// TimeZone
fbSpecificLocalTime(in := Tc2_Utilities.FILETIME64_TO_SYSTEMTIME(fbEvent.nTimestamp), tzInfo := fbTimeZone.tzInfo, out => _TempTimestruct);

// Timestamp	
THIS^.stEventInfo.TimeRaised[0] := TO_DINT(_TempTimestruct.wYear);
THIS^.stEventInfo.TimeRaised[1] := TO_DINT(_TempTimestruct.wMonth);
THIS^.stEventInfo.TimeRaised[2] := TO_DINT(_TempTimestruct.wDay);
THIS^.stEventInfo.TimeRaised[3] := TO_DINT(_TempTimestruct.wHour);
THIS^.stEventInfo.TimeRaised[4] := TO_DINT(_TempTimestruct.wMinute);
THIS^.stEventInfo.TimeRaised[5] := TO_DINT(_TempTimestruct.wSecond);
THIS^.stEventInfo.TimeRaised[6] := TO_DINT(_TempTimestruct.wMilliseconds);
Tc2_System.MEMSET(destAddr := ADR(stEventInfo.TimeCleared), fillByte := 0, n := SIZEOF(stEventInfo.TimeCleared));
Tc2_System.MEMSET(destAddr := ADR(stEventInfo.TimeConfirmed), fillByte := 0, n := SIZEOF(stEventInfo.TimeConfirmed));

//store event info globally
aEventInfoBuffer[CntAlarmsRaised] := stEventInfo;

// activate requests in event triggered method 'OnMessageSent' to get related request info
aEventInfoBuffer[CntAlarmsRaised].fbRequestEventText.Request(eventClass := aEventInfoBuffer[CntAlarmsRaised].EventClass,
															 nEventId	:= aEventInfoBuffer[CntAlarmsRaised].EventId,
															 nLangId	:= 1033,
															 ipArgs		:= aEventInfoBuffer[CntAlarmsRaised].ipArguments);

OnAlarmRaised := S_OK; // in order to receive more callbacks (Set <> S_OK in order to cancel the callbacks for this program cycle.)
END_METHOD

PROPERTY ParentResponseDefinitions : ARRAY[0..4] OF SPT_BaseTypes.E_AlarmResponse
GET
ParentResponseDefinitions := _ParentResponseDefinitions;
END_GET
SET
_ParentResponseDefinitions := ParentResponseDefinitions;
END_SET
END_PROPERTY

METHOD Reset : BOOL
//This may or may not be called depending on the component type 

//which derives FB_ComponentBase
F_ClearAllEventsInClass(PackMLEventHandlerAlarms);
Reset := TRUE;
END_METHOD

METHOD PUBLIC TimeZone : BOOL
VAR_INST
	_Step : USINT; // Step Variable
END_VAR
CASE _Step OF
	0: // Start to get local Timezone 
		fbTimeZone.bExecute := TRUE;
		IF fbTimeZone.bBusy THEN
			_Step := _Step + 1;
		END_IF

	1: // set 
		fbTimeZone.bExecute := FALSE;
		_Step				:= 0;
		TimeZone			:= TRUE;

ELSE
	Tc2_System.ADSLOGSTR(msgCtrlMask := cMsgCtrlMask, msgFmtStr := Tc2_Standard.CONCAT(cBaseMsg, 'TimeZone: %s'), strArg := 'Case Idx error');
	_InternalError := TRUE;
END_CASE

fbTimeZone(sNetID := '');
IF fbTimeZone.bError THEN
	Tc2_System.ADSLOGSTR(msgCtrlMask := cMsgCtrlMask, msgFmtStr := Tc2_Standard.CONCAT(cBaseMsg, 'fbTimeZone ErrID: %s'), strArg := TO_STRING(fbTimeZone.nErrID));
	_InternalError := TRUE;
END_IF
END_METHOD

PROPERTY WarningToStopReason : BOOL
SET
_WarningToStopReason := WarningToStopReason;
END_SET
END_PROPERTY

METHOD PRIVATE WriteAlarmTags : HRESULT;
VAR_INPUT
	Alarm_Ref	  : REFERENCE TO Tc3_PackML_V2.ST_Alarm; // Reference to ST_Alarm of an new Alarm / Warning / Stop reason
	EventInfo_Ref : REFERENCE TO ST_EventInfo;			 // Reference to ST_EventInfo
	Trigger		  : BOOL;								 // Set / Reset Trigger in PML Structure
	AlarmIndex	  : DINT;								 // Alarm index
END_VAR
IF __ISVALIDREF(Alarm_Ref) AND __ISVALIDREF(EventInfo_Ref) THEN
	Alarm_Ref.ID	   := TO_DINT(EventInfo_Ref.EventId);
	Alarm_Ref.Value	   := AlarmIndex;
	Alarm_Ref.Message  := EventInfo_Ref.EventText;
	Alarm_Ref.Category := TO_DINT(EventInfo_Ref.eSeverity); // Verbose:=0, Info:=1, Warning:=2, Error:=3, Critical:=4
	Alarm_Ref.Trigger  := Trigger;
	Alarm_Ref.DateTime := EventInfo_Ref.TimeRaised;
	WriteAlarmTags	   := S_OK;
ELSE
	// Set internal Error
	Tc2_System.ADSLOGSTR(msgCtrlMask := cMsgCtrlMask, msgFmtStr := Tc2_Standard.CONCAT(cBaseMsg, 'WriteAlarmTags: %s'), strArg := 'Input-reference error');
	WriteAlarmTags := E_FAIL;
	_InternalError := TRUE;
END_IF
END_METHOD

END_FUNCTION_BLOCK

// Project Information/F_GetCompany
// This function has been automatically generated from the project information.
{attribute 'signature_flag' := '1073741824'}
{attribute 'TcGenerated'}
{attribute 'no-analysis'}
FUNCTION F_GetCompany : WSTRING
VAR_INPUT
	
END_VAR

F_GetCompany := "Beckhoff Automation LLC";

END_FUNCTION

// Project Information/F_GetTitle
// This function has been automatically generated from the project information.
{attribute 'signature_flag' := '1073741824'}
{attribute 'TcGenerated'}
{attribute 'no-analysis'}
FUNCTION F_GetTitle : WSTRING
VAR_INPUT
	
END_VAR

F_GetTitle := "SPT Components";

END_FUNCTION

// Project Information/F_GetVersion
// This function has been automatically generated from the project information.
{attribute 'signature_flag' := '1073741824'}
{attribute 'TcGenerated'}
{attribute 'no-analysis'}
FUNCTION F_GetVersion : ST_LibVersion
VAR_INPUT
	
END_VAR

F_GetVersion.iMajor := 3;
F_GetVersion.iMinor := 2;
F_GetVersion.iBuild := 3;
F_GetVersion.iRevision := 0;
F_GetVersion.sVersion := '3.2.3';
F_GetVersion.nFlags := 1;

END_FUNCTION

// Sensors/FB_DigitalSensor
FUNCTION_BLOCK FB_DigitalSensor EXTENDS FB_ComponentBase IMPLEMENTS I_DigitalSensorBase
VAR
	HardwareInput AT %I*		: BOOL;			  //Hardware input bit from the hysical sensor
	_DebounceMode				: E_DebounceMode; //Defines the debounce model that will filter the sensor's output to the program
	_DebounceTime				: TIME;			  //Time input parameter for use in Debounce functionality
	_Inverted					: BOOL;			  //Defines the output polarity of the sensor - a "TRUE" value will result in the signal of the sensor being inverted
	_SimulationInput			: BOOL;			  //Provides configuration input to the simulation functionality
	_SimulationTimebase			: UDINT;
	_SimulationMode				: E_SensorSimulationMode; //Defines the mode of operation for the simulation functionality of this component
	_TimeActive					: TIME;					  //Tracks the amount of time that the sensor has been in an active state
	_TimeInactive				: TIME;					  //Tracks the amount of time that the sensor has been in an inactive state
	_Active						: BOOL;
	TON_ActiveTimer				: Tc2_Standard.TON; //Tracks the amount of time that the sensor has been in an active state
	TON_InactiveTimer			: Tc2_Standard.TON; //Tracks the amount of time that the sensor has been in an inactive state
	TON_DebounceTimer			: Tc2_Standard.TON; //Utilized in the debounce implementation
	TP_DebounceTimer			: Tc2_Standard.TP;	//Utilized in the debounce implementation
	DigitalSensor_HMI			: ST_DigitalSensor_HMI;
	SimulationPulse1_TP			: Tc2_Standard.TP; //Pulse Timer for simulated sensor pulse generation
	SimulationPulse2_TP			: Tc2_Standard.TP; //Pulse Timer for simulated sensor pulse generation
	HMICommand_DigitalSensor_RT : R_TRIG;
END_VAR

METHOD PUBLIC CyclicLogic
VAR_INPUT
END_VAR
SUPER^.CyclicLogic();
IF _Simulate THEN
	CASE _SimulationMode OF
		E_SensorSimulationMode.InputDriven:
			_Active := _SimulationInput;

		E_SensorSimulationMode.Periodic:
			SimulationPulse1_TP(IN := NOT SimulationPulse2_TP.Q, PT := UDINT_TO_TIME(_SimulationTimebase));
			SimulationPulse2_TP(IN := NOT SimulationPulse1_TP.Q, PT := UDINT_TO_TIME(_SimulationTimebase));
			_Active := SimulationPulse2_TP.Q;
	END_CASE
ELSE
	_Active := ProcessInput(Input := HardwareInput);
END_IF
END_METHOD

PROPERTY Active : BOOL
GET
Active := _Active;
END_GET
END_PROPERTY

PROPERTY DebounceMode : E_DebounceMode
GET
DebounceMode := _DebounceMode;
END_GET
SET
_DebounceMode := DebounceMode;
END_SET
END_PROPERTY

PROPERTY DebounceTime : TIME
GET
DebounceTime := _DebounceTime;
END_GET
SET
_DebounceTime := DebounceTime;
END_SET
END_PROPERTY

PROPERTY Inverted : BOOL
GET
Inverted := _Inverted;
END_GET
SET
_Inverted := Inverted;
END_SET
END_PROPERTY

PROPERTY SimulationInput : BOOL
GET
SimulationInput := _SimulationInput;
END_GET
SET
_SimulationInput := SimulationInput;
END_SET
END_PROPERTY

PROPERTY SimulationMode : E_SensorSimulationMode
GET
SimulationMode := _SimulationMode;
END_GET
SET
_SimulationMode := SimulationMode;
END_SET
END_PROPERTY

PROPERTY SimulationTimeBase : UDINT
GET
SimulationTimeBase := _SimulationTimebase;
END_GET
SET
_SimulationTimeBase := SimulationTimebase;
END_SET
END_PROPERTY

PROPERTY TimeActive : TIME
GET
TimeActive := _TimeActive;
END_GET
END_PROPERTY

PROPERTY TimeInactive : TIME
GET
TimeInactive := _TimeInactive;
END_GET
END_PROPERTY

METHOD PROTECTED HMICommunication
//Extend this method in extended FBs to communicate specific implementation data
SUPER^.HMICommunication();

//Process HMI requests

//Replace 'FALSE' below with further momentary commands (myCommand XOR myOtherCommand XOR...)
HMICommand_DigitalSensor_RT(CLK := (ComponentBase_HMI.Status.HMIControlAvailable AND NOT HMICommandActive_Base) AND (FALSE));

//Signal to FB_ComponentBase that a command is active
HMICommandActive_Descendant := ComponentBase_HMI.Status.HMIControlAvailable AND (DigitalSensor_HMI.Config.DebounceMode <> _DebounceMode OR DigitalSensor_HMI.Config.DebounceTime <> _DebounceTime OR DigitalSensor_HMI.Config.Inverted <> _Inverted OR DigitalSensor_HMI.Config.SimulationMode <> _SimulationMode OR DigitalSensor_HMI.Config.SimulationTimebase <> _SimulationTimebase);

//Process HMI requests
IF HMICommand_DigitalSensor_RT.Q THEN //If a request has been issued by the HMI, and a previous request has not just finished being processed

	//	IF AxisBaseHMI.Command.xxx THEN

	//		Enabled := TRUE;

	//	END_IF
END_IF

IF ComponentBase_HMI.Status.HMIControlAvailable AND NOT HMICommand_DigitalSensor_RT.Q THEN
	IF DigitalSensor_HMI.Config.DebounceMode <> _DebounceMode THEN
		DebounceMode := DigitalSensor_HMI.Config.DebounceMode;
	END_IF

	IF DigitalSensor_HMI.Config.DebounceTime <> _DebounceTime THEN
		DebounceTime := DigitalSensor_HMI.Config.DebounceTime;
	END_IF

	IF DigitalSensor_HMI.Config.Inverted <> _Inverted THEN
		Inverted := DigitalSensor_HMI.Config.Inverted;
	END_IF

	IF DigitalSensor_HMI.Config.SimulationMode <> _SimulationMode THEN
		SimulationMode := DigitalSensor_HMI.Config.SimulationMode;
	END_IF

	IF DigitalSensor_HMI.Config.SimulationTimebase <> _SimulationTimebase THEN
		SimulationTimeBase := DigitalSensor_HMI.Config.SimulationTimebase;
	END_IF
END_IF

//Update HMI status info
DigitalSensor_HMI.Status.Active				:= _Active;
DigitalSensor_HMI.Status.TimeActive			:= TIME_TO_LREAL(_TimeActive) / 1000.0;
DigitalSensor_HMI.Status.TimeInactive		:= TIME_TO_LREAL(_TimeInactive) / 1000.0;
DigitalSensor_HMI.Config.DebounceMode		:= DebounceMode;
DigitalSensor_HMI.Config.DebounceTime		:= DebounceTime;
DigitalSensor_HMI.Config.Inverted			:= Inverted;
DigitalSensor_HMI.Config.SimulationMode		:= SimulationMode;
DigitalSensor_HMI.Config.SimulationTimebase := SimulationTimeBase;
END_METHOD

METHOD PROTECTED Monitoring
SUPER^.Monitoring();

//If flicker counters or other diagnostic systems are desired, their implementation could be here

//Any warnings, errors, or other desired messages would also be generated here

//T#71582M47S295MS is the upper bound of the TIME type, meaning these timers will continue to increase ET for as long as possible
TON_ActiveTimer(IN := _Active, PT := T#71582M47S295MS, ET => _TimeActive);
TON_InactiveTimer(IN := NOT _Active, PT := T#71582M47S295MS, ET => _TimeInactive);
_Busy  := FALSE;
_Error := FALSE;
END_METHOD

METHOD PRIVATE ProcessInput : BOOL
VAR_INPUT
	Input : BOOL;
END_VAR

VAR
	DebouncedInput : BOOL;
END_VAR

VAR_INST
	LastDebouncedInput : BOOL;
	MovingAverage	   : DINT;
END_VAR
CASE DebounceMode OF
	E_DebounceMode.RawInput: //Passes raw input through
		DebouncedInput := Input;

	E_DebounceMode.SimpleFlickerFilter:											 //Requires the raw input to be a consistent value for a set time period before output changes
		TON_DebounceTimer(IN := (Input <> DebouncedInput), PT := _DebounceTime); //runs the timer whenever a differing input is detected
		IF TON_DebounceTimer.Q THEN
			DebouncedInput := Input; //once the raw input has been different for the specified debounce time, the processed input is updated
		END_IF

	E_DebounceMode.EdgeDetectFilter:								   //Updates the processed value immediately on a change from steady state, but mutes any sensor flickers for the specified time immediately following the change
		IF (Input <> DebouncedInput) AND (NOT TP_DebounceTimer.Q) THEN //A differing raw input must be detected outside of the mute window created by the pulse timer
			DebouncedInput := Input;
		END_IF

		TP_DebounceTimer(IN := (DebouncedInput <> LastDebouncedInput), PT := _DebounceTime); //"Q" will be TRUE for tDebounce time after the bProcessedSensorInput value is changed
	E_DebounceMode.MovingAverage:															 //Uses a "moving average"-like calculation to compensate for extremely inconsistent signals - prevents poorly timed flickers from causing disproportionate results
		TON_DebounceTimer(IN := NOT TON_DebounceTimer.Q, PT := T#5MS);						 //Provides a 1ms "polling" trigger
		IF TON_DebounceTimer.Q THEN															 //TRUE once every millisecond
			IF Input THEN																	 //If raw input is currently active at the time of polling
				IF MovingAverage < TIME_TO_DINT(_DebounceTime) THEN							 //If the moving average has not reached its "weight limit" as set by debounce time
					MovingAverage := MovingAverage + 5;										 //Add 1 to the average
				END_IF
			ELSE													 //If raw input is currently inactive at the time of polling
				IF MovingAverage > -TIME_TO_DINT(_DebounceTime) THEN //If the moving average has not reached its "weight limit" as set by debounce time
					MovingAverage := MovingAverage - 5;				 //Subtract 1 from the average
				END_IF
			END_IF
		END_IF

		IF MovingAverage >= 0 THEN
			DebouncedInput := TRUE;
		ELSE
			DebouncedInput := FALSE;
		END_IF
END_CASE

LastDebouncedInput := DebouncedInput; //Update "Last value"
IF _Inverted THEN					  //If signal inversion is requested, invert the signal
	DebouncedInput := NOT DebouncedInput;
END_IF

ProcessInput := DebouncedInput;
END_METHOD

END_FUNCTION_BLOCK

// Sensors/I_DigitalSensorBase
INTERFACE I_DigitalSensorBase

PROPERTY DebounceMode : E_DebounceMode
GET
END_GET
SET
END_SET
END_PROPERTY

PROPERTY DebounceTime : TIME
GET
END_GET
SET
END_SET
END_PROPERTY

PROPERTY Inverted : BOOL //"High" signal from the sensor will be interpreted as an "inactive" reading when this parameter is TRUE
GET
END_GET
SET
END_SET
END_PROPERTY

PROPERTY SimulationInput : BOOL
GET
END_GET
SET
END_SET
END_PROPERTY

PROPERTY SimulationMode : E_SensorSimulationMode
GET
END_GET
SET
END_SET
END_PROPERTY

PROPERTY TimeActive : TIME
GET
END_GET
END_PROPERTY

PROPERTY TimeInactive : TIME
GET
END_GET
END_PROPERTY

END_INTERFACE

// Solenoids/SolenoidBankBase/FB_SolenoidBankBase
FUNCTION_BLOCK ABSTRACT FB_SolenoidBankBase EXTENDS FB_ComponentBase
VAR
	// Configuration
	Configuration : ARRAY[1..Parameters_Cylinder.MAX_NUMBER_OF_SOLENOIDS] OF ST_SolenoidBankConfig;

	//Counted number of solenoids
	NumberOfSolenoids : UINT;

	//Alarms
	SolenoidBankAlarms : ARRAY[1..SolenoidBankBaseAlarmsCount] OF FB_TcAlarm;
END_VAR

VAR CONSTANT
	SolenoidBankBaseAlarmsCount : UINT := 2;
END_VAR

METHOD PUBLIC AddSolenoid : UINT
VAR_INPUT
	ipCylinder	 : I_Solenoid;
	Number		 : UINT; //This is the number in the IO tree.
	SolenoidType : E_SolenoidType;
END_VAR
IF CheckNumber(Number) AND ipCylinder <> 0 THEN
	NumberOfSolenoids									  := NumberOfSolenoids + 1;
	Configuration[NumberOfSolenoids].ipSolenoid			  := ipCylinder;
	Configuration[NumberOfSolenoids].SolenoidType		  := SolenoidType;
	Configuration[NumberOfSolenoids].SolenoidOutputNumber := Number;
END_IF
END_METHOD

METHOD PRIVATE CheckNumber : BOOL
VAR_INPUT
	Number : UINT;
END_VAR
CheckNumber := TRUE;
IF Number < 1 AND Number > Parameters_Cylinder.MAX_NUMBER_OF_SOLENOIDS THEN
	IF NOT SolenoidBankAlarms[E_CylinderBankAlarms.CylinderNumberOutOfRange].bRaised THEN
		SolenoidBankAlarms[E_CylinderBankAlarms.CylinderNumberOutOfRange].Raise(0);
	END_IF

	CheckNumber := FALSE;
END_IF
END_METHOD

//! @summary Initializes event function blocks using this components's name
{attribute 'call_after_online_change_slot' := '<slot>'}
METHOD PROTECTED CreateEvents

//! @description This method is called by <c>Initialize()</c> as required
SUPER^.CreateEvents();
F_CreateAllEventsInClass(Alarms		:= SolenoidBankAlarms,
						 ClassSize	:= SIZEOF(TC_EVENTS.CylinderBankAlarms),
						 pInitEvent := ADR(TC_EVENTS.CylinderBankAlarms.InitReferenceEvent),
						 Prefix		:= Name);
END_METHOD

//! @summary This method serves as the entry point for all underlying FB logic
METHOD PUBLIC CyclicLogic
//! @description This method should be called cyclically by descendant function blocks by invoking <c>SUPER^.CyclicLogic()</c>.  Alternatively, the contents of this method could be reimplemented entirely in which case a call to this method would not be necessary.
VAR
	x : UINT;
END_VAR
//Loop through all solenoids that are added.
FOR x := 1 TO NumberOfSolenoids DO
	MapIO(x);
END_FOR
END_METHOD

//! @summary Basic component initialization logic
METHOD PROTECTED Initialize : BOOL;
//! @description This method is called by <c>CyclicLogic()</c> as required
VAR
	x : UINT;
END_VAR
NumberOfSolenoids := 0;
Initialize		  := TRUE;
END_METHOD

METHOD ABSTRACT MapIO
VAR_INPUT
	x : UINT;
END_VAR
END_METHOD

//! Provides basic error detection and event handling for this component
METHOD PROTECTED Monitoring

(*! @descriptionThis method is called cyclically by <c>CyclicLogic()</c>*)
SUPER^.Monitoring();
_CurrentAlarmSeverity := F_GetMaxSeverityRaised(Alarms := SolenoidBankAlarms, CurrentSeverity := CurrentAlarmSeverity);
END_METHOD

//! @summary Clears error flags and error IDs for this component
METHOD PUBLIC Reset : BOOL
SUPER^.Reset();
IF SolenoidBankAlarms[E_CylinderBankAlarms.CylinderNumberOutOfRange].bRaised THEN
	SolenoidBankAlarms[E_CylinderBankAlarms.CylinderNumberOutOfRange].Clear(0, 0);
END_IF
END_METHOD

END_FUNCTION_BLOCK

// Solenoids/I_Solenoid
INTERFACE I_Solenoid

METHOD Extend
VAR_INPUT
END_VAR
END_METHOD

PROPERTY Extended : BOOL
GET
END_GET
END_PROPERTY

PROPERTY ExtendOutput : BOOL
GET
END_GET
END_PROPERTY

PROPERTY ExtendTime : LREAL
GET
END_GET
SET
END_SET
END_PROPERTY

METHOD Retract
VAR_INPUT
END_VAR
END_METHOD

PROPERTY Retracted : BOOL
GET
END_GET
END_PROPERTY

PROPERTY RetractOutput : BOOL
GET
END_GET
END_PROPERTY

PROPERTY RetractTime : LREAL
GET
END_GET
SET
END_SET
END_PROPERTY

END_INTERFACE

// Solenoids/FB_DoubleSolenoid
FUNCTION_BLOCK FB_DoubleSolenoid EXTENDS FB_SingleSolenoid
VAR
	_RetractOutput AT %Q* : BOOL;
END_VAR

METHOD PROTECTED HardwareInit
//Update the status based on the IO 
IF _ExtendOutput AND NOT _RetractOutput THEN
	_Extended  := TRUE;
	_Retracted := FALSE;
ELSIF NOT _ExtendOutput AND _RetractOutput THEN
	_Extended  := FALSE;
	_Retracted := TRUE;
ELSE // By Default, set RetractOuptupt if neither is set or if both are set.
	_ExtendOutput  := FALSE;
	_RetractOutput := TRUE;
	_Extended	   := FALSE;
	_Retracted	   := TRUE;
END_IF
END_METHOD

METHOD PROTECTED HardwareUpdate
//One shot the requests
Extend_RTRIG(CLK := _ExtendRequest);
Retract_RTRIG(CLK := _RetractRequest);

//Handle Extend
IF Extend_RTRIG.Q THEN
	_ExtendOutput	:= TRUE;
	_RetractOutput	:= FALSE;
	_Extending		:= TRUE;
	_Retracting		:= FALSE;
	_Retracted		:= FALSE;
	_RetractRequest := FALSE;
END_IF

//Handle Retract
IF Retract_RTRIG.Q THEN
	_ExtendOutput  := FALSE;
	_RetractOutput := TRUE;
	_Extending	   := FALSE;
	_Retracting	   := TRUE;
	_Extended	   := FALSE;
	_ExtendRequest := FALSE;
END_IF

//Always Simulate Feedback here with no feedback inputs
Feedback();
END_METHOD

PROPERTY RetractOutput : BOOL
GET
RetractOutput := _RetractOutput;
END_GET
END_PROPERTY

END_FUNCTION_BLOCK

// Solenoids/FB_SingleSolenoid
(*	This FB is used for a single output solenoid 
	It uses the times to say when Extended/Retracted  	
	It starts assuming retracted and the output off.
*)
FUNCTION_BLOCK FB_SingleSolenoid EXTENDS FB_ComponentBase IMPLEMENTS I_Solenoid
VAR
	//Output
	_ExtendOutput AT %Q* : BOOL;

	// Internal variables
	_ExtendRequest	: BOOL;
	_RetractRequest : BOOL;
	_Extended		: BOOL;
	_Retracted		: BOOL;
	_Extending		: BOOL;
	_Retracting		: BOOL;
	_ExtendTime		: LREAL := 1000; // Default time 1s
	_RetractTime	: LREAL := 1000; // Default time 1s

	// Timer for Extend/Retract
	Extend_TON	  : TON;
	Retract_TON	  : TON;
	Extend_RTRIG  : R_TRIG;
	Retract_RTRIG : R_TRIG;

	//HMI 
	SolenoidHMI : ST_Cylinder_HMI;

	//Alarms
	SolenoidAlarms : ARRAY[1..SolenoidAlarmsCount] OF FB_TcAlarm;
END_VAR

VAR CONSTANT
	SolenoidAlarmsCount : UINT := 4;
END_VAR

METHOD PROTECTED CreateEvents
VAR_INPUT
END_VAR
SUPER^.CreateEvents();
F_CreateAllEventsInClass(Alarms		:= SolenoidAlarms,
						 ClassSize	:= SIZEOF(TC_EVENTS.CylinderAlarms),
						 pInitEvent := ADR(TC_EVENTS.CylinderAlarms.InitReferenceEvent),
						 Prefix		:= Name);
END_METHOD

METHOD PROTECTED HMICommunication
VAR_INPUT
END_VAR
SUPER^.HMICommunication();

//Handle the requests to extend and retract
IF ComponentBase_HMI.Status.HMIControlAvailable THEN
	IF SolenoidHMI.Command.Extend THEN
		Extend();
	ELSIF SolenoidHMI.Command.Retract THEN
		Retract();
	END_IF

	IF NOT F_CompareLREAL(SolenoidHMI.Command.ExtendTime, _ExtendTime, 0.01) THEN
		_ExtendTime := SolenoidHMI.Command.ExtendTime;
	END_IF

	IF NOT F_CompareLREAL(SolenoidHMI.Command.RetractTime, _RetractTime, 0.01) THEN
		_RetractTime := SolenoidHMI.Command.RetractTime;
	END_IF
END_IF

//Update HMI status info
SolenoidHMI.Status.Extended	   := _Extended;
SolenoidHMI.Status.Extending   := _Extending;
SolenoidHMI.Status.Retracted   := _Retracted;
SolenoidHMI.Status.Retracting  := _Retracting;
SolenoidHMI.Config.ExtendTime  := _ExtendTime;
SolenoidHMI.Config.RetractTime := _RetractTime;
END_METHOD

METHOD PROTECTED Monitoring
VAR_INPUT
END_VAR
SUPER^.Monitoring();

//Update output bits
_Busy				  := _Extending OR _Retracting;
_CurrentAlarmSeverity := F_GetMaxSeverityRaised(Alarms := SolenoidAlarms, CurrentSeverity := CurrentAlarmSeverity);
_Error				  := _CurrentAlarmSeverity >= TcEventSeverity.Error;
END_METHOD

METHOD CyclicLogic
VAR
	myErrorID : UDINT;
END_VAR
HardwareUpdate();
SUPER^.CyclicLogic();

//New code
myErrorID := THIS^.ErrorID;
END_METHOD

METHOD Extend
_ExtendRequest	:= TRUE;
_RetractRequest := FALSE;
END_METHOD

PROPERTY Extended : BOOL
GET
Extended := _Extended;
END_GET
END_PROPERTY

PROPERTY ExtendOutput : BOOL
GET
ExtendOutput := _ExtendOutput;
END_GET
END_PROPERTY

PROPERTY ExtendTime : LREAL
GET
ExtendTime := _ExtendTime;
END_GET
SET
_ExtendTime					   := ExtendTime;
SolenoidHMI.Command.ExtendTime := ExtendTime;
END_SET
END_PROPERTY

METHOD Retract
_ExtendRequest	:= FALSE;
_RetractRequest := TRUE;
END_METHOD

PROPERTY Retracted : BOOL
GET
Retracted := _Retracted;
END_GET
END_PROPERTY

PROPERTY RetractOutput : BOOL
GET
RetractOutput := FALSE;
END_GET
END_PROPERTY

PROPERTY RetractTime : LREAL
GET
RetractTime := _RetractTime;
END_GET
SET
_RetractTime					:= RetractTime;
SolenoidHMI.Command.RetractTime := RetractTime;
END_SET
END_PROPERTY

METHOD PROTECTED Feedback
VAR_INPUT
END_VAR
//Handle the time to Extend/Retract
Extend_TON(IN := _Extending, PT := LREAL_TO_TIME(_ExtendTime));
Retract_TON(IN := _Retracting, PT := LREAL_TO_TIME(_RetractTime));
IF Extend_TON.Q THEN
	_Extended  := TRUE;
	_Extending := FALSE;
END_IF

IF Retract_TON.Q THEN
	_Retracted	:= TRUE;
	_Retracting := FALSE;
END_IF
END_METHOD

METHOD PROTECTED HardwareInit
IF _ExtendOutput THEN
	_Extended  := TRUE;
	_Retracted := FALSE;
ELSE
	_Extended  := FALSE;
	_Retracted := TRUE;
END_IF
END_METHOD

METHOD PROTECTED HardwareUpdate
VAR_INPUT
END_VAR
//One shot the requests
Extend_RTRIG(CLK := _ExtendRequest);
Retract_RTRIG(CLK := _RetractRequest);

//Handle Extend
IF Extend_RTRIG.Q THEN
	_ExtendOutput	:= TRUE;
	_Extending		:= TRUE;
	_Retracting		:= FALSE;
	_Retracted		:= FALSE;
	_RetractRequest := FALSE;
END_IF

//Handle Retract
IF Retract_RTRIG.Q THEN
	_ExtendOutput  := FALSE;
	_Extending	   := FALSE;
	_Retracting	   := TRUE;
	_Extended	   := FALSE;
	_ExtendRequest := FALSE;
END_IF

//Call the feedback 
Feedback();
END_METHOD

//! @summary Basic component initialization logic
METHOD PROTECTED Initialize : BOOL;

//! @description This method is called by <c>CyclicLogic()</c> as required
//Set the cylinder to retracted
_Extending		:= FALSE;
_ExtendRequest	:= FALSE;
_Retracting		:= FALSE;
_RetractRequest := FALSE;

//Set the HMI time to the currnt time.
SolenoidHMI.Command.ExtendTime	:= _ExtendTime;
SolenoidHMI.Command.RetractTime := _RetractTime;

//Call base class Initialize
Initialize := SUPER^.Initialize();

// Call the HardwareInit
HardwareInit();
END_METHOD

//! @summary Clears error flags and error IDs for this component
METHOD PUBLIC Reset : BOOL
Reset := FALSE;
F_ClearAllEventsInClass(Alarms := SolenoidAlarms);
END_METHOD

END_FUNCTION_BLOCK

// Solenoids/FB_DoubleSolenoidFeedback
FUNCTION_BLOCK FB_DoubleSolenoidFeedback EXTENDS FB_DoubleSolenoid
VAR
	ExtendedSensor	AT %I* : BOOL;
	RetractedSensor AT %I* : BOOL;
END_VAR

PROPERTY ExtendedInput : BOOL
SET
ExtendedSensor := ExtendedInput;
END_SET
END_PROPERTY

METHOD PROTECTED Feedback
IF NOT _Simulate THEN
	_Extended  := ExtendedSensor;
	_Retracted := RetractedSensor;
	Extend_TON(IN := _Extending, PT := LREAL_TO_TIME(_ExtendTime));
	Retract_TON(IN := _Retracting, PT := LREAL_TO_TIME(_RetractTime));
	IF Extend_TON.Q AND NOT ExtendedSensor THEN
		IF NOT SolenoidAlarms[E_CylinderAlarms.ExtendTimeout].bRaised THEN
			SolenoidAlarms[E_CylinderAlarms.ExtendTimeout].Raise(0);
			_ExtendRequest := FALSE;
			_Extending	   := FALSE;
		END_IF
	ELSIF _Extending AND ExtendedSensor THEN
		_Extended  := TRUE;
		_Extending := FALSE;
	END_IF

	IF Retract_TON.Q AND NOT RetractedSensor THEN
		IF NOT SolenoidAlarms[E_CylinderAlarms.RetractTimeout].bRaised THEN
			SolenoidAlarms[E_CylinderAlarms.RetractTimeout].Raise(0);
			_RetractRequest := FALSE;
			_Retracting		:= FALSE;
		END_IF
	ELSIF _Retracting AND RetractedSensor THEN
		_Retracted	:= TRUE;
		_Retracting := FALSE;
	END_IF
ELSE
	SUPER^.Feedback();
END_IF

//Monitor Inputs in case both on at the same time
IF ExtendedSensor AND RetractedSensor AND NOT SolenoidAlarms[E_CylinderAlarms.ExtendedAndRetracted].bRaised THEN
	SolenoidAlarms[E_CylinderAlarms.ExtendedAndRetracted].Raise(0);
ELSIF (ExtendedSensor XOR RetractedSensor) AND SolenoidAlarms[E_CylinderAlarms.ExtendedAndRetracted].bRaised THEN
	SolenoidAlarms[E_CylinderAlarms.ExtendedAndRetracted].Clear(0, 0);
END_IF
END_METHOD

METHOD PROTECTED HardwareInit
IF ExtendedSensor AND NOT RetractedSensor THEN
	_Extended  := TRUE;
	_Retracted := FALSE;
ELSIF NOT ExtendedSensor AND RetractedSensor THEN
	_Extended  := FALSE;
	_Retracted := TRUE;
ELSE // With Neither on, then this means that it is not either or maybe no air
	_Extended  := FALSE;
	_Retracted := FALSE;
END_IF
END_METHOD

PROPERTY RetractedInput : BOOL
SET
RetractedSensor := RetractedInput;
END_SET
END_PROPERTY

END_FUNCTION_BLOCK

// Solenoids/FB_SingleSolenoidFeedback
FUNCTION_BLOCK FB_SingleSolenoidFeedback EXTENDS FB_SingleSolenoid
VAR
	ExtendedSensor	AT %I* : BOOL;
	RetractedSensor AT %I* : BOOL;
END_VAR

PROPERTY ExtendedInput : BOOL
SET
ExtendedSensor := ExtendedInput;
END_SET
END_PROPERTY

METHOD PROTECTED Feedback
IF NOT _Simulate THEN
	_Extended  := ExtendedSensor;
	_Retracted := RetractedSensor;
	Extend_TON(IN := _Extending, PT := LREAL_TO_TIME(_ExtendTime));
	Retract_TON(IN := _Retracting, PT := LREAL_TO_TIME(_RetractTime));
	IF Extend_TON.Q AND NOT ExtendedSensor THEN
		IF NOT SolenoidAlarms[E_CylinderAlarms.ExtendTimeout].bRaised THEN
			SolenoidAlarms[E_CylinderAlarms.ExtendTimeout].Raise(0);
			_ExtendRequest := FALSE;
			_Extending	   := FALSE;
		END_IF
	ELSIF _Extending AND ExtendedSensor THEN
		_Extended  := TRUE;
		_Extending := FALSE;
	END_IF

	IF Retract_TON.Q AND NOT RetractedSensor THEN
		IF NOT SolenoidAlarms[E_CylinderAlarms.RetractTimeout].bRaised THEN
			SolenoidAlarms[E_CylinderAlarms.RetractTimeout].Raise(0);
			_RetractRequest := FALSE;
			_Retracting		:= FALSE;
		END_IF
	ELSIF _Retracting AND RetractedSensor THEN
		_Retracted	:= TRUE;
		_Retracting := FALSE;
	END_IF
ELSE
	SUPER^.Feedback(); //Call the feedback that usese timers for feedback
END_IF

//Monitor Inputs in case both on at the same time
IF ExtendedSensor AND RetractedSensor AND NOT SolenoidAlarms[E_CylinderAlarms.ExtendedAndRetracted].bRaised THEN
	SolenoidAlarms[E_CylinderAlarms.ExtendedAndRetracted].Raise(0);
ELSIF (ExtendedSensor XOR RetractedSensor) AND SolenoidAlarms[E_CylinderAlarms.ExtendedAndRetracted].bRaised THEN
	SolenoidAlarms[E_CylinderAlarms.ExtendedAndRetracted].Clear(0, 0);
END_IF
END_METHOD

METHOD PROTECTED HardwareInit
IF ExtendedSensor AND NOT RetractedSensor THEN
	_Extended  := TRUE;
	_Retracted := FALSE;
ELSIF NOT ExtendedSensor AND RetractedSensor THEN
	_Extended  := FALSE;
	_Retracted := TRUE;
ELSE // With Neither on, then this means that it is not either or maybe no air
	_Extended  := FALSE;
	_Retracted := FALSE;
END_IF
END_METHOD

PROPERTY RetractedInput : BOOL
SET
RetractedSensor := RetractedInput;
END_SET
END_PROPERTY

END_FUNCTION_BLOCK

// Testing/Axis/FB_ComponentBasicAxis_Test
FUNCTION_BLOCK FB_ComponentBasicAxis_Test EXTENDS TCUnit.FB_TestSuite
VAR
	TestFBInit					: FB_Component_BasicAxis;
	TestFBNameSetProperty		: FB_Component_BasicAxis;
	TestFBSimulationSetProperty : FB_Component_BasicAxis;
	TestFBSimulationSetHMI		: FB_Component_BasicAxis;
	TestFBSimulationCheckAlarm	: FB_Component_BasicAxis;
	TestFBBusy					: FB_Component_BasicAxis;
	TestFBAllowHMI				: FB_Component_BasicAxis;
	TestFBBlockHMI				: FB_Component_BasicAxis;

	//Axis integration test - this should be tested in the NCAxis library. (Enable, Disable, etc....)

	//Alarm Testing - 17 Alarms with FB_ComponentBasicAxis

	///TestFBAlarm1  FB_Component_BasicAxis; // InitReference (Not an actual alarm)
	TestFBAlarm2 : FB_Component_BasicAxis; // MC_Power
	TestFBAlarm3 : FB_Component_BasicAxis; // MC_Reset
	TestFBAlarm4 : FB_Component_BasicAxis; // MC_Halt

	///TestFBAlarm5 FB_Component_BasicAxis; // MC_Stop // Not Implemented
	TestFBAlarm6  : FB_Component_BasicAxis; // MC_Home
	TestFBAlarm7  : FB_Component_BasicAxis; // MC_Jog
	TestFBAlarm8  : FB_Component_BasicAxis; // MC_MoveAbsolute
	TestFBAlarm9  : FB_Component_BasicAxis; // MC_MoveRelative
	TestFBAlarm10 : FB_Component_BasicAxis; // MC_MoveVelocity
	TestFBAlarm11 : FB_Component_BasicAxis; // MC_MoveModulo
	TestFBAlarm12 : FB_Component_BasicAxis; // MC_ReadParameter
	TestFBAlarm13 : FB_Component_BasicAxis; // MC_WriteParameter
	TestFBAlarm14 : FB_Component_BasicAxis; // MC_WriteBOOLParameter
	TestFBAlarm15 : FB_Component_BasicAxis; // Command While Inhibited

	///TestFBAlarm16 FB_Component_BasicAxis; // Axis Error (Not Sure how to get Axis error with virtual axis)

	///TestFBAlarm17 FB_Component_BasicAxis; // Drive Error (Cannot Get Drive Error without drive)
END_VAR

Init();
NameSetProperty();
SimulationSetProperty();
SimulationSetHMI();
SimulationCheckAlarm();
Busy();
AllowHMI();
BlockHMI();

//Tests for Alarms
MCPowerAlarm();
MCResetAlarm();
MCHaltAlarm();
MCHomeAlarm();
MCJogAlarm();
MCMoveAbsoluteAlarm();
MCMoveRelativeAlarm();
MCMoveVelocity();
MCMoveModulo();
McReadAxisParametersAlarm();
McWriteAxisParameterAlarm();
McWriteAxisBoolParameterAlarm();
CommandInhibited();

METHOD AllowHMI
VAR_INST
	State		   : INT;
	ActualResult   : BOOL;
	ExpectedResult : BOOL := TRUE;
END_VAR
IF TEST_ORDERED('BasicAxisAllowHMI') THEN
	CASE State OF
		0:
			State := State + 10;

		10:
			IF TestFBAllowHMI.InitComplete AND NOT TestFBAllowHMI.Busy THEN
				TestFBAllowHMI.AllowHMIControl();
				State := State + 10;
			END_IF

		20:
			ActualResult := TestFBAllowHMI.ComponentBase_HMI.Status.HMIControlAvailable;
			AssertEquals_BOOL(Expected := ExpectedResult, Actual := ActualResult, Message := 'Function Block read allow HMI Control in HMI Tag not true');
			TEST_FINISHED();
			State := State + 10;
	END_CASE

	//Call to FB Cyclic Logic
	TestFBAllowHMI.CyclicLogic();
END_IF
END_METHOD

METHOD BlockHMI
VAR_INST
	State		   : INT;
	ActualResult   : BOOL;
	ExpectedResult : BOOL := FALSE;
END_VAR
IF TEST_ORDERED('BasicAxisBlockHMI') THEN
	CASE State OF
		0:
			State := State + 10;

		10:
			IF TestFBBlockHMI.InitComplete AND NOT TestFBBlockHMI.Busy THEN
				TestFBBlockHMI.AllowHMIControl();
				State := State + 10;
			END_IF

		20:
			IF TestFBBlockHMI.ComponentBase_HMI.Status.HMIControlAvailable THEN
				TestFBBlockHMI.BlockHMIControl();
				State := State + 10;
			END_IF

		30:
			ActualResult := TestFBBlockHMI.ComponentBase_HMI.Status.HMIControlAvailable;
			AssertEquals_BOOL(Expected := ExpectedResult, Actual := ActualResult, Message := 'Function Block read Block HMI Control in HMI Tag not false');
			TEST_FINISHED();
			State := State + 10;
	END_CASE

	//Call to FB Cyclic Logic
	TestFBBlockHMI.CyclicLogic();
END_IF
END_METHOD

METHOD Busy
VAR_INST
	State		   : INT;
	ActualResult   : BOOL;
	ExpectedResult : BOOL := TRUE;
	Timeout		   : TON;
END_VAR
IF TEST_ORDERED('BasicAxisBusy') THEN
	CASE State OF
		0:
			State := State + 10;

		10:
			IF TestFBBusy.InitComplete AND NOT TestFBBusy.Busy THEN
				TestFBBusy.Enable();
				State := State + 10;
			END_IF

		20:
			IF TestFBBusy.Enabled THEN
				TestFBBusy.Acceleration := 1000;
				TestFBBusy.Deceleration := 1000;
				TestFBBusy.Velocity		:= 100;
				TestFBBusy.MoveAbsolute(100, TRUE);
				State := State + 10;
			END_IF

		30:
			ActualResult := TestFBBusy.Busy;
			AssertEquals_BOOL(Expected := ExpectedResult, Actual := ActualResult, Message := 'Function Block was not busy when Extending');
			TEST_FINISHED();
			State := State + 10;
	END_CASE

	//Call to FB Cyclic Logic
	TestFBBusy.CyclicLogic();
END_IF
END_METHOD

METHOD CommandInhibited
VAR_INST
	State		   : INT;
	ActualResult   : BOOL;
	ExpectedResult : BOOL := TRUE;
END_VAR
IF TEST_ORDERED('CommandInhibitedAlarm') THEN
	CASE State OF
		0:
			IF TestFBAlarm15.InitComplete THEN
				TestFBAlarm15.Override := 0;
				TestFBAlarm15.MoveAbsolute(100, TRUE);
				State := State + 10;
			END_IF

		10:
			IF TestFBAlarm15.Error OR (TestFBAlarm15.InPosition AND NOT TestFBAlarm15.Busy) THEN
				ActualResult := TestFBAlarm15.BasicAxisAlarms[E_BasicAxis.CommandWhileInhibited].bRaised;
				State		 := State + 10;
			END_IF

		20:
			AssertEquals_BOOL(Expected := ExpectedResult, Actual := ActualResult, Message := 'The alarm was not raised for Command Inhibited Error');
			TEST_FINISHED();
			State := State + 10;
	END_CASE

	TestFBAlarm15.CyclicLogic();
END_IF
END_METHOD

METHOD Init
VAR_INST
	State		   : INT;
	ActualResult   : BOOL;
	ExpectedResult : BOOL := TRUE;
	Timeout		   : TON;
END_VAR
IF TEST_ORDERED('BasicAxisInit') THEN
	CASE State OF
		0:
			Timeout.IN := TRUE;
			State	   := State + 10;

		10:
			IF TestFBInit.InitComplete AND NOT TestFBInit.Busy THEN
				State := State + 10;
			END_IF

			IF Timeout.Q THEN
				State := State + 10;
			END_IF

		20:
			ActualResult := TestFBInit.InitComplete;
			AssertEquals_BOOL(Expected := ExpectedResult, Actual := ActualResult, Message := 'Function Block did not init complete in 2s');
			TEST_FINISHED();
			State := State + 10;
	END_CASE

	//Call to FB Cyclic Logic
	Timeout(PT := T#2S);
	TestFBInit.CyclicLogic();
END_IF
END_METHOD

METHOD MCHaltAlarm
VAR_INST
	State		   : INT;
	ActualResult   : BOOL;
	ExpectedResult : BOOL := TRUE;
	WriteADS	   : FB_WriteAdsSymByName;
END_VAR
IF TEST_ORDERED('MCHaltAlarm') THEN
	CASE State OF
		0:
			WriteADS(bWrite	  := TRUE,
					 sNetId	  := '',
					 nPort	  := 851,
					 sVarName := 'PRG_TEST.ComponentBasicAxisTest.TestFBAlarm4.BasicAxis.MCHalt.Error',
					 nSrcAddr := ADR(ExpectedResult),
					 nLen	  := SIZEOF(ExpectedResult),
					 tTimeout := T#2S,
					 eComMode :=,
					 bBusy	  =>,
					 bError	  =>,
					 nErrorId =>);

			IF NOT WriteADS.bBusy OR WriteADS.bError THEN
				State := State + 10;
			END_IF

			IF TestFBAlarm4.BasicAxisAlarms[E_BasicAxis.HaltError].bRaised THEN
				ActualResult := TestFBAlarm4.BasicAxisAlarms[E_BasicAxis.HaltError].bRaised;
				State		 := State + 10;
			END_IF

		10:
			AssertEquals_BOOL(Expected := ExpectedResult, Actual := ActualResult, Message := 'The alarm was not raised for MC_Halt.Error');
			TEST_FINISHED();
			State := State + 10;
	END_CASE

	TestFBAlarm4.CyclicLogic();
END_IF
END_METHOD

METHOD MCHomeAlarm
VAR_INST
	State		   : INT;
	ActualResult   : BOOL;
	ExpectedResult : BOOL := TRUE;
	WriteADS	   : FB_WriteAdsSymByName;
END_VAR
IF TEST_ORDERED('MCHomeAlarm') THEN
	CASE State OF
		0:
			WriteADS(bWrite	  := TRUE,
					 sNetId	  := '',
					 nPort	  := 851,
					 sVarName := 'PRG_TEST.ComponentBasicAxisTest.TestFBAlarm6.BasicAxis.DefaultHome._Error',
					 nSrcAddr := ADR(ExpectedResult),
					 nLen	  := SIZEOF(ExpectedResult),
					 tTimeout := T#2S,
					 eComMode :=,
					 bBusy	  =>,
					 bError	  =>,
					 nErrorId =>);

			IF NOT WriteADS.bBusy OR WriteADS.bError THEN
				State := State + 10;
			END_IF

			IF TestFBAlarm6.BasicAxisAlarms[E_BasicAxis.HomeError].bRaised THEN
				ActualResult := TestFBAlarm6.BasicAxisAlarms[E_BasicAxis.HomeError].bRaised;
				State		 := State + 10;
			END_IF

		10:
			AssertEquals_BOOL(Expected := ExpectedResult, Actual := ActualResult, Message := 'The alarm was not raised for HomeMethod.Error');
			TEST_FINISHED();
			State := State + 10;
	END_CASE

	TestFBAlarm6.CyclicLogic();
END_IF
END_METHOD

METHOD MCJogAlarm
VAR_INST
	State		   : INT;
	ActualResult   : BOOL;
	ExpectedResult : BOOL := TRUE;
	WriteADS	   : FB_WriteAdsSymByName;
END_VAR
IF TEST_ORDERED('MCJogAlarm') THEN
	CASE State OF
		0:
			WriteADS(bWrite	  := TRUE,
					 sNetId	  := '',
					 nPort	  := 851,
					 sVarName := 'PRG_TEST.ComponentBasicAxisTest.TestFBAlarm7.BasicAxis.MCJog.Error',
					 nSrcAddr := ADR(ExpectedResult),
					 nLen	  := SIZEOF(ExpectedResult),
					 tTimeout := T#2S,
					 eComMode :=,
					 bBusy	  =>,
					 bError	  =>,
					 nErrorId =>);

			IF NOT WriteADS.bBusy OR WriteADS.bError THEN
				State := State + 10;
			END_IF

			IF TestFBAlarm7.BasicAxisAlarms[E_BasicAxis.JogError].bRaised THEN
				ActualResult := TestFBAlarm7.BasicAxisAlarms[E_BasicAxis.JogError].bRaised;
				State		 := State + 10;
			END_IF

		10:
			AssertEquals_BOOL(Expected := ExpectedResult, Actual := ActualResult, Message := 'The alarm was not raised for MCJog.Error');
			TEST_FINISHED();
			State := State + 10;
	END_CASE

	TestFBAlarm7.CyclicLogic();
END_IF
END_METHOD

METHOD MCMoveAbsoluteAlarm
VAR_INST
	State		   : INT;
	ActualResult   : BOOL;
	ExpectedResult : BOOL := TRUE;
END_VAR
IF TEST_ORDERED('MCMoveAbsAlarm') THEN
	CASE State OF
		0:
			IF TestFBAlarm8.InitComplete THEN
				TestFBAlarm8.MoveAbsolute(100, TRUE);
				State := State + 10;
			END_IF

		10:
			IF TestFBAlarm8.Error OR (TestFBAlarm8.InPosition AND NOT TestFBAlarm8.Busy) THEN
				State := State + 10;
			END_IF

		20:
			ActualResult := TestFBAlarm8.BasicAxisAlarms[E_BasicAxis.MoveAbsoluteError].bRaised;
			AssertEquals_BOOL(Expected := ExpectedResult, Actual := ActualResult, Message := 'The alarm was not raised for Move Absolute Error');
			TEST_FINISHED();
			State := State + 10;
	END_CASE

	TestFBAlarm8.CyclicLogic();
END_IF
END_METHOD

METHOD MCMoveModulo
VAR_INST
	State		   : INT;
	ActualResult   : BOOL;
	ExpectedResult : BOOL := TRUE;
END_VAR
IF TEST_ORDERED('MCMoveModuloAlarm') THEN
	CASE State OF
		0:
			IF TestFBAlarm11.InitComplete THEN
				TestFBAlarm11.MoveModulo(100, MC_Direction.MC_Positive_Direction, TRUE);
				State := State + 10;
			END_IF

		10:
			IF TestFBAlarm11.Error OR (TestFBAlarm11.InPosition AND NOT TestFBAlarm11.Busy) THEN
				State := State + 10;
			END_IF

		20:
			ActualResult := TestFBAlarm11.BasicAxisAlarms[E_BasicAxis.MoveModuloError].bRaised;
			AssertEquals_BOOL(Expected := ExpectedResult, Actual := ActualResult, Message := 'The alarm was not raised for Move Modulo Error');
			TEST_FINISHED();
			State := State + 10;
	END_CASE

	TestFBAlarm11.CyclicLogic();
END_IF
END_METHOD

METHOD MCMoveRelativeAlarm
VAR_INST
	State		   : INT;
	ActualResult   : BOOL;
	ExpectedResult : BOOL := TRUE;
END_VAR
IF TEST_ORDERED('MCMoveAbsAlarm') THEN
	CASE State OF
		0:
			IF TestFBAlarm9.InitComplete THEN
				TestFBAlarm9.MoveRelative(100, TRUE);
				State := State + 10;
			END_IF

		10:
			IF TestFBAlarm9.Error OR (TestFBAlarm9.InPosition AND NOT TestFBAlarm9.Busy) THEN
				State := State + 10;
			END_IF

		20:
			ActualResult := TestFBAlarm9.BasicAxisAlarms[E_BasicAxis.MoveRelativeError].bRaised;
			AssertEquals_BOOL(Expected := ExpectedResult, Actual := ActualResult, Message := 'The alarm was not raised for Move Relative Error');
			TEST_FINISHED();
			State := State + 10;
	END_CASE

	TestFBAlarm9.CyclicLogic();
END_IF
END_METHOD

METHOD MCMoveVelocity
VAR_INST
	State		   : INT;
	ActualResult   : BOOL;
	ExpectedResult : BOOL := TRUE;
END_VAR
IF TEST_ORDERED('MCMoveVelAlarm') THEN
	CASE State OF
		0:
			IF TestFBAlarm10.InitComplete THEN
				TestFBAlarm10.MoveVelocity(100, TRUE);
				State := State + 10;
			END_IF

		10:
			IF TestFBAlarm10.Error OR (TestFBAlarm10.InPosition AND NOT TestFBAlarm10.Busy) THEN
				State := State + 10;
			END_IF

		20:
			ActualResult := TestFBAlarm10.BasicAxisAlarms[E_BasicAxis.MoveVelocityError].bRaised;
			AssertEquals_BOOL(Expected := ExpectedResult, Actual := ActualResult, Message := 'The alarm was not raised for Move Relative Error');
			TEST_FINISHED();
			State := State + 10;
	END_CASE

	TestFBAlarm10.CyclicLogic();
END_IF
END_METHOD

METHOD MCPowerAlarm
VAR_INST
	State		   : INT;
	ActualResult   : BOOL;
	ExpectedResult : BOOL := TRUE;
	WriteADS	   : FB_WriteAdsSymByName;
END_VAR
IF TEST_ORDERED('MCPowerAlarm') THEN
	CASE State OF
		0:
			WriteADS(bWrite	  := TRUE,
					 sNetId	  := '',
					 nPort	  := 851,
					 sVarName := 'PRG_TEST.ComponentBasicAxisTest.TestFBAlarm2.BasicAxis.MCPower.Error',
					 nSrcAddr := ADR(ExpectedResult),
					 nLen	  := SIZEOF(ExpectedResult),
					 tTimeout := T#2S,
					 eComMode :=,
					 bBusy	  =>,
					 bError	  =>,
					 nErrorId =>);

			IF NOT WriteADS.bBusy OR WriteADS.bError THEN
				State := State + 10;
			END_IF

			IF TestFBAlarm2.BasicAxisAlarms[E_BasicAxis.PowerError].bRaised THEN
				ActualResult := TestFBAlarm2.BasicAxisAlarms[E_BasicAxis.PowerError].bRaised;
				State		 := State + 10;
			END_IF

		10:
			AssertEquals_BOOL(Expected := ExpectedResult, Actual := ActualResult, Message := 'The alarm was not raised for MC_Power.Error');
			TEST_FINISHED();
			State := State + 10;
	END_CASE

	TestFBAlarm2.CyclicLogic();
END_IF
END_METHOD

METHOD McReadAxisParametersAlarm
VAR_INST
	State		   : INT;
	ActualResult   : BOOL;
	ExpectedResult : BOOL := TRUE;
	WriteADS	   : FB_WriteAdsSymByName;
END_VAR
IF TEST_ORDERED('MCReadAxisAlarm') THEN
	CASE State OF
		0:
			WriteADS(bWrite	  := TRUE,
					 sNetId	  := '',
					 nPort	  := 851,
					 sVarName := 'PRG_TEST.ComponentBasicAxisTest.TestFBAlarm12.BasicAxis.MCReadParameterSet.Error',
					 nSrcAddr := ADR(ExpectedResult),
					 nLen	  := SIZEOF(ExpectedResult),
					 tTimeout := T#2S,
					 eComMode :=,
					 bBusy	  =>,
					 bError	  =>,
					 nErrorId =>);

			IF NOT WriteADS.bBusy OR WriteADS.bError THEN
				State := State + 10;
			END_IF

			IF TestFBAlarm12.BasicAxisAlarms[E_BasicAxis.ReadParameterSetError].bRaised THEN
				ActualResult := TestFBAlarm12.BasicAxisAlarms[E_BasicAxis.ReadParameterSetError].bRaised;
				State		 := State + 10;
			END_IF

		10:
			AssertEquals_BOOL(Expected := ExpectedResult, Actual := ActualResult, Message := 'The alarm was not raised for MC Read Axis Parameter Error');
			TEST_FINISHED();
			State := State + 10;
	END_CASE

	TestFBAlarm12.CyclicLogic();
END_IF
END_METHOD

METHOD MCResetAlarm
VAR_INST
	State		   : INT;
	ActualResult   : BOOL;
	ExpectedResult : BOOL := TRUE;
	WriteADS	   : FB_WriteAdsSymByName;
END_VAR
IF TEST_ORDERED('MCResetAlarm') THEN
	CASE State OF
		0:
			WriteADS(bWrite	  := TRUE,
					 sNetId	  := '',
					 nPort	  := 851,
					 sVarName := 'PRG_TEST.ComponentBasicAxisTest.TestFBAlarm3.BasicAxis.DefaultReset._Error',
					 nSrcAddr := ADR(ExpectedResult),
					 nLen	  := SIZEOF(ExpectedResult),
					 tTimeout := T#2S,
					 eComMode :=,
					 bBusy	  =>,
					 bError	  =>,
					 nErrorId =>);

			IF NOT WriteADS.bBusy OR WriteADS.bError THEN
				State := State + 10;
			END_IF

			IF TestFBAlarm3.BasicAxisAlarms[E_BasicAxis.ResetError].bRaised THEN
				ActualResult := TestFBAlarm3.BasicAxisAlarms[E_BasicAxis.ResetError].bRaised;
				State		 := State + 10;
			END_IF

		10:
			AssertEquals_BOOL(Expected := ExpectedResult, Actual := ActualResult, Message := 'The alarm was not raised for ResetMethod.Error');
			TEST_FINISHED();
			State := State + 10;
	END_CASE

	TestFBAlarm3.CyclicLogic();
END_IF
END_METHOD

METHOD McWriteAxisBoolParameterAlarm
VAR_INST
	State		   : INT;
	ActualResult   : BOOL;
	ExpectedResult : BOOL := TRUE;
	WriteADS	   : FB_WriteAdsSymByName;
END_VAR
IF TEST_ORDERED('MCWriteAxisBoolAlarm') THEN
	CASE State OF
		0:
			WriteADS(bWrite	  := TRUE,
					 sNetId	  := '',
					 nPort	  := 851,
					 sVarName := 'PRG_TEST.ComponentBasicAxisTest.TestFBAlarm14.BasicAxis.MCWriteBoolParameter.Error',
					 nSrcAddr := ADR(ExpectedResult),
					 nLen	  := SIZEOF(ExpectedResult),
					 tTimeout := T#2S,
					 eComMode :=,
					 bBusy	  =>,
					 bError	  =>,
					 nErrorId =>);

			IF NOT WriteADS.bBusy OR WriteADS.bError THEN
				State := State + 10;
			END_IF

			IF TestFBAlarm14.BasicAxisAlarms[E_BasicAxis.WriteBoolParameterError].bRaised THEN
				ActualResult := TestFBAlarm14.BasicAxisAlarms[E_BasicAxis.WriteBoolParameterError].bRaised;
				State		 := State + 10;
			END_IF

		10:
			AssertEquals_BOOL(Expected := ExpectedResult, Actual := ActualResult, Message := 'The alarm was not raised for MC Write Axis Bool Parameter Error');
			TEST_FINISHED();
			State := State + 10;
	END_CASE

	TestFBAlarm14.CyclicLogic();
END_IF
END_METHOD

METHOD McWriteAxisParameterAlarm
VAR_INST
	State		   : INT;
	ActualResult   : BOOL;
	ExpectedResult : BOOL := TRUE;
	WriteADS	   : FB_WriteAdsSymByName;
END_VAR
IF TEST_ORDERED('MCWriteAxisAlarm') THEN
	CASE State OF
		0:
			WriteADS(bWrite	  := TRUE,
					 sNetId	  := '',
					 nPort	  := 851,
					 sVarName := 'PRG_TEST.ComponentBasicAxisTest.TestFBAlarm13.BasicAxis.MCWriteParameter.Error',
					 nSrcAddr := ADR(ExpectedResult),
					 nLen	  := SIZEOF(ExpectedResult),
					 tTimeout := T#2S,
					 eComMode :=,
					 bBusy	  =>,
					 bError	  =>,
					 nErrorId =>);

			IF NOT WriteADS.bBusy OR WriteADS.bError THEN
				State := State + 10;
			END_IF

			IF TestFBAlarm13.BasicAxisAlarms[E_BasicAxis.WriteParameterError].bRaised THEN
				ActualResult := TestFBAlarm13.BasicAxisAlarms[E_BasicAxis.WriteParameterError].bRaised;
				State		 := State + 10;
			END_IF

		10:
			AssertEquals_BOOL(Expected := ExpectedResult, Actual := ActualResult, Message := 'The alarm was not raised for MC Write Axis Parameter Error');
			TEST_FINISHED();
			State := State + 10;
	END_CASE

	TestFBAlarm13.CyclicLogic();
END_IF
END_METHOD

METHOD NameSetProperty
VAR_INST
	State			: INT;
	ActualResult	: STRING;
	ActualResultHMI : STRING;
	ExpectedResult	: STRING := 'TEST_NAME';
END_VAR
IF TEST_ORDERED('BasicAxisNameSetProperty') THEN
	CASE State OF
		0:
			State := State + 10;

		10:
			IF TestFBNameSetProperty.InitComplete AND NOT TestFBNameSetProperty.Busy THEN
				State := State + 10;
			END_IF

		20:
			TestFBNameSetProperty.Name := ExpectedResult;
			State					   := State + 10;

		30:
			ActualResultHMI := TestFBNameSetProperty.ComponentBase_HMI.Config.Name;
			ActualResult	:= TestFBNameSetProperty.Name;
			AssertEquals(Expected := ExpectedResult, Actual := ActualResult, Message := 'Name was not read by Property correctly');
			AssertEquals(Expected := ExpectedResult, Actual := ActualResultHMI, Message := 'Name was not read by HMI correctly');
			TEST_FINISHED();
			State := State + 10;
	END_CASE

	//Call to FB Cyclic Logic
	TestFBNameSetProperty.CyclicLogic();
END_IF
END_METHOD

METHOD SimulationCheckAlarm
VAR_INST
	State		   : INT;
	ActualResult   : BOOL;
	ExpectedResult : BOOL := TRUE;
END_VAR
IF TEST_ORDERED('BasicAxisSimulationCheckAlarm') THEN
	CASE State OF
		0:
			State := State + 10;

		10:
			IF TestFBSimulationCheckAlarm.InitComplete AND NOT TestFBSimulationCheckAlarm.Busy THEN
				State := State + 10;
			END_IF

		20:
			TestFBSimulationCheckAlarm.InSimulation := TRUE; //Set simulation to true;
			State									:= State + 10;

		30:
			ActualResult := TestFBSimulationCheckAlarm.ComponentBaseAlarms[E_ComponentBase.SimulationWarning].bRaised;
			AssertEquals_BOOL(Expected := ExpectedResult, Actual := ActualResult, Message := 'Function Block did Raise alarm when in simulation');
			TEST_FINISHED();
			State := State + 10;
	END_CASE

	//Call to FB Cyclic Logic
	TestFBSimulationCheckAlarm.CyclicLogic();
END_IF
END_METHOD

METHOD SimulationSetHMI
VAR_INST
	State			: INT;
	ActualResult	: BOOL;
	ActualResultHMI : BOOL;
	ExpectedResult	: BOOL := TRUE;
	WriteADS		: FB_WriteAdsSymByName;
END_VAR
IF TEST_ORDERED('BasicAxisSetSimulationHMI') THEN
	CASE State OF
		0:
			State := State + 10;

		10:
			IF TestFBSimulationSetHMI.InitComplete AND NOT TestFBSimulationSetHMI.Busy THEN
				TestFBSimulationSetHMI.AllowHMIControl(); // Must turn on Allow control for code to function
				State := State + 10;
			END_IF

		20:
			WriteADS(bWrite	  := TRUE,
					 sNetId	  := '',
					 nPort	  := 851,
					 sVarName := 'PRG_TEST.ComponentBasicAxisTest.TestFBSimulationSetHMI.ComponentBase_HMI.Command.SimulatedOperation',
					 nSrcAddr := ADR(ExpectedResult),
					 nLen	  := SIZEOF(ExpectedResult),
					 tTimeout := T#2S,
					 eComMode :=,
					 bBusy	  =>,
					 bError	  =>,
					 nErrorId =>);

			IF NOT WriteADS.bBusy OR WriteADS.bError THEN
				State := State + 10;
			END_IF

		30:
			ActualResult	:= TestFBSimulationSetHMI.InSimulation;
			ActualResultHMI := TestFBSimulationSetHMI.ComponentBase_HMI.Status.InSimulation;
			AssertEquals_BOOL(Expected := ExpectedResult, Actual := ActualResult, Message := 'Function Block did not set simulation by HMI when read by Property');
			AssertEquals_BOOL(Expected := ExpectedResult, Actual := ActualResultHMI, Message := 'Function Block did not set simulation by HMI when read by HMI');
			TEST_FINISHED();
			State := State + 10;
	END_CASE

	//Call to FB Cyclic Logic
	TestFBSimulationSetHMI.CyclicLogic();
END_IF
END_METHOD

METHOD SimulationSetProperty
VAR_INST
	State			: INT;
	ActualResult	: BOOL;
	ActualResultHMI : BOOL;
	ExpectedResult	: BOOL := TRUE;
END_VAR
IF TEST_ORDERED('BasicAxisSetSimulationProperty') THEN
	CASE State OF
		0:
			State := State + 10;

		10:
			IF TestFBSimulationSetProperty.InitComplete AND NOT TestFBSimulationSetProperty.Busy THEN
				State := State + 10;
			END_IF

		20:
			TestFBSimulationSetProperty.InSimulation := TRUE;
			State									 := State + 10;

		30:
			ActualResult	:= TestFBSimulationSetProperty.InSimulation;
			ActualResultHMI := TestFBSimulationSetProperty.ComponentBase_HMI.Status.InSimulation;
			AssertEquals_BOOL(Expected := ExpectedResult, Actual := ActualResult, Message := 'Function Block did not set simulation by property when read by Property');
			AssertEquals_BOOL(Expected := ExpectedResult, Actual := ActualResultHMI, Message := 'Function Block did not set simulation by property when read by HMI');
			TEST_FINISHED();
			State := State + 10;
	END_CASE

	//Call to FB Cyclic Logic
	TestFBSimulationSetProperty.CyclicLogic();
END_IF
END_METHOD

END_FUNCTION_BLOCK

// Testing/PRG_TEST
PROGRAM PRG_TEST
VAR
	SingleSolenoidTest		   : FB_SingleSolenoid_Test;
	DoubleSolenoidTest		   : FB_DoubleSolenoid_Test;
	SingleSolenoidFeedbackTest : FB_SingleSolenoidFeedback_Test;
	ComponentBasicAxisTest	   : FB_ComponentBasicAxis_Test;
END_VAR

TcUnit.RUN();

END_PROGRAM

// Testing/Solenoids/FB_SingleSolenoid_Test
FUNCTION_BLOCK FB_SingleSolenoid_Test EXTENDS TcUnit.FB_TestSuite
VAR
	// FBs for ComponentBase
	TestFBInit					: FB_SingleSolenoid;
	TestFBNameSetProperty		: FB_SingleSolenoid;
	TestFBNameSetHMI			: FB_SingleSolenoid;
	TestFBSimulationSetProperty : FB_SingleSolenoid;
	TestFBSimulationSetHMI		: FB_SingleSolenoid;
	TestFBSimulationCheckAlarm	: FB_SingleSolenoid;
	TestFBBusy					: FB_SingleSolenoid;
	TestFBAllowHMI				: FB_SingleSolenoid;
	TestFBBlockHMI				: FB_SingleSolenoid;

	// Solenoid FB	
	TestSingleSolenoidExtend  : FB_SingleSolenoid;
	TestSingleSolenoidRetract : FB_SingleSolenoid;
END_VAR

Init();
NameSetProperty();
SimulationSetProperty();
SimulationSetHMI();
SimulationCheckAlarm();
Busy();
AllowHMI();
BlockHMI();
ExtendEqualsExtendedOutputOn();
RetractEqualsExtendOutputOff();

METHOD AllowHMI
VAR_INST
	State		   : INT;
	ActualResult   : BOOL;
	ExpectedResult : BOOL := TRUE;
END_VAR
IF TEST_ORDERED('AllowHMI') THEN
	CASE State OF
		0:
			State := State + 10;

		10:
			IF TestFBAllowHMI.InitComplete AND NOT TestFBAllowHMI.Busy THEN
				TestFBAllowHMI.AllowHMIControl();
				State := State + 10;
			END_IF

		20:
			ActualResult := TestFBAllowHMI.ComponentBase_HMI.Status.HMIControlAvailable;
			AssertEquals_BOOL(Expected := ExpectedResult, Actual := ActualResult, Message := 'Function Block read allow HMI Control in HMI Tag not true');
			TEST_FINISHED();
			State := State + 10;
	END_CASE

	//Call to FB Cyclic Logic
	TestFBAllowHMI.CyclicLogic();
END_IF
END_METHOD

METHOD BlockHMI
VAR_INST
	State		   : INT;
	ActualResult   : BOOL;
	ExpectedResult : BOOL := FALSE;
END_VAR
IF TEST_ORDERED('BlockHMI') THEN
	CASE State OF
		0:
			State := State + 10;

		10:
			IF TestFBBlockHMI.InitComplete AND NOT TestFBBlockHMI.Busy THEN
				TestFBBlockHMI.AllowHMIControl();
				State := State + 10;
			END_IF

		20:
			IF TestFBBlockHMI.ComponentBase_HMI.Status.HMIControlAvailable THEN
				TestFBBlockHMI.BlockHMIControl();
				State := State + 10;
			END_IF

		30:
			ActualResult := TestFBBlockHMI.ComponentBase_HMI.Status.HMIControlAvailable;
			AssertEquals_BOOL(Expected := ExpectedResult, Actual := ActualResult, Message := 'Function Block read Block HMI Control in HMI Tag not false');
			TEST_FINISHED();
			State := State + 10;
	END_CASE

	//Call to FB Cyclic Logic
	TestFBBlockHMI.CyclicLogic();
END_IF
END_METHOD

METHOD Busy
VAR_INST
	State		   : INT;
	ActualResult   : BOOL;
	ExpectedResult : BOOL := TRUE;
	Timeout		   : TON;
END_VAR
IF TEST_ORDERED('Busy') THEN
	CASE State OF
		0:
			State := State + 10;

		10:
			IF TestFBBusy.InitComplete AND NOT TestFBBusy.Busy THEN
				State := State + 10;
			END_IF

		20:
			TestFBBusy.Extend();
			State := State + 10;

		30:
			ActualResult := TestFBBusy.Busy;
			AssertEquals_BOOL(Expected := ExpectedResult, Actual := ActualResult, Message := 'Function Block was not busy when Extending');
			TEST_FINISHED();
			State := State + 10;
	END_CASE

	//Call to FB Cyclic Logic
	TestFBBusy.CyclicLogic();
END_IF
END_METHOD

METHOD ExtendEqualsExtendedOutputOn
VAR_INST
	State		   : INT;
	ActualResult   : BOOL;
	ExpectedResult : BOOL := TRUE;
END_VAR
IF TEST_ORDERED('ExtendEqualsExtendedOutputOn') THEN
	CASE State OF
		0:
			State := State + 10;

		10:
			TestSingleSolenoidExtend.Extend();
			State := State + 10;

		20:
			ActualResult := TestSingleSolenoidExtend.ExtendOutput;
			AssertEquals_BOOL(Expected := ExpectedResult, Actual := ActualResult, Message := 'Solenoid did not set output on');
			TEST_FINISHED();
			State := State + 10;
	END_CASE

	TestSingleSolenoidExtend.CyclicLogic();
END_IF
END_METHOD

METHOD Init
VAR_INST
	State		   : INT;
	ActualResult   : BOOL;
	ExpectedResult : BOOL := TRUE;
	Timeout		   : TON;
END_VAR
IF TEST_ORDERED('Init') THEN
	CASE State OF
		0:
			Timeout.IN := TRUE;
			State	   := State + 10;

		10:
			IF TestFBInit.InitComplete AND NOT TestFBInit.Busy THEN
				State := State + 10;
			END_IF

			IF Timeout.Q THEN
				State := State + 10;
			END_IF

		20:
			ActualResult := TestFBInit.InitComplete;
			AssertEquals_BOOL(Expected := ExpectedResult, Actual := ActualResult, Message := 'Function Block did not init complete in 2s');
			TEST_FINISHED();
			State := State + 10;
	END_CASE

	//Call to FB Cyclic Logic
	Timeout(PT := T#2S);
	TestFBInit.CyclicLogic();
END_IF
END_METHOD

METHOD NameSetProperty
VAR_INST
	State			: INT;
	ActualResult	: STRING;
	ActualResultHMI : STRING;
	ExpectedResult	: STRING := 'TEST_NAME';
END_VAR
IF TEST_ORDERED('NameSetProperty') THEN
	CASE State OF
		0:
			State := State + 10;

		10:
			IF TestFBNameSetProperty.InitComplete AND NOT TestFBNameSetProperty.Busy THEN
				State := State + 10;
			END_IF

		20:
			TestFBNameSetProperty.Name := ExpectedResult;
			State					   := State + 10;

		30:
			ActualResultHMI := TestFBNameSetProperty.ComponentBase_HMI.Config.Name;
			ActualResult	:= TestFBNameSetProperty.Name;
			AssertEquals(Expected := ExpectedResult, Actual := ActualResult, Message := 'Name was not read by Property correctly');
			AssertEquals(Expected := ExpectedResult, Actual := ActualResultHMI, Message := 'Name was not read by HMI correctly');
			TEST_FINISHED();
			State := State + 10;
	END_CASE

	//Call to FB Cyclic Logic
	TestFBNameSetProperty.CyclicLogic();
END_IF
END_METHOD

METHOD RetractEqualsExtendOutputOff
VAR_INST
	State		   : INT;
	ActualResult   : BOOL;
	ExpectedResult : BOOL := FALSE;
END_VAR
IF TEST_ORDERED('RetractEqualsExtendOutputOff') THEN
	CASE State OF
		0:
			State := State + 10;

		10:
			TestSingleSolenoidRetract.Retract();
			State := State + 10;

		20:
			ActualResult := TestSingleSolenoidRetract.ExtendOutput;
			AssertEquals_BOOL(Expected := ExpectedResult, Actual := ActualResult, Message := 'Solenoid did not set output on');
			TEST_FINISHED();
			State := State + 10;
	END_CASE

	TestSingleSolenoidRetract.CyclicLogic();
END_IF
END_METHOD

METHOD SimulationCheckAlarm
VAR_INST
	State		   : INT;
	ActualResult   : BOOL;
	ExpectedResult : BOOL := TRUE;
END_VAR
IF TEST_ORDERED('SimulationCheckAlarm') THEN
	CASE State OF
		0:
			State := State + 10;

		10:
			IF TestFBSimulationCheckAlarm.InitComplete AND NOT TestFBSimulationCheckAlarm.Busy THEN
				State := State + 10;
			END_IF

		20:
			TestFBSimulationCheckAlarm.InSimulation := TRUE; //Set simulation to true;
			State									:= State + 10;

		30:
			ActualResult := TestFBSimulationCheckAlarm.ComponentBaseAlarms[E_ComponentBase.SimulationWarning].bRaised;
			AssertEquals_BOOL(Expected := ExpectedResult, Actual := ActualResult, Message := 'Function Block did Raise alarm when in simulation');
			TEST_FINISHED();
			State := State + 10;
	END_CASE

	//Call to FB Cyclic Logic
	TestFBSimulationCheckAlarm.CyclicLogic();
END_IF
END_METHOD

METHOD SimulationSetHMI
VAR_INST
	State			: INT;
	ActualResult	: BOOL;
	ActualResultHMI : BOOL;
	ExpectedResult	: BOOL := TRUE;
	WriteADS		: FB_WriteAdsSymByName;
END_VAR
IF TEST_ORDERED('SimulationSetHMI') THEN
	CASE State OF
		0:
			State := State + 10;

		10:
			IF TestFBSimulationSetHMI.InitComplete AND NOT TestFBSimulationSetHMI.Busy THEN
				TestFBSimulationSetHMI.AllowHMIControl(); // Must turn on Allow control for code to function
				State := State + 10;
			END_IF

		20:
			WriteADS(bWrite	  := TRUE,
					 sNetId	  := '',
					 nPort	  := 851,
					 sVarName := 'PRG_TEST.SingleSolenoidTest.TestFBSimulationSetHMI.ComponentBase_HMI.Command.SimulatedOperation',
					 nSrcAddr := ADR(ExpectedResult),
					 nLen	  := SIZEOF(ExpectedResult),
					 tTimeout := T#2S,
					 eComMode :=,
					 bBusy	  =>,
					 bError	  =>,
					 nErrorId =>);

			IF NOT WriteADS.bBusy OR WriteADS.bError THEN
				State := State + 10;
			END_IF

		30:
			ActualResult	:= TestFBSimulationSetHMI.InSimulation;
			ActualResultHMI := TestFBSimulationSetHMI.ComponentBase_HMI.Status.InSimulation;
			AssertEquals_BOOL(Expected := ExpectedResult, Actual := ActualResult, Message := 'Function Block did not set simulation by HMI when read by Property');
			AssertEquals_BOOL(Expected := ExpectedResult, Actual := ActualResultHMI, Message := 'Function Block did not set simulation by HMI when read by HMI');
			TEST_FINISHED();
			State := State + 10;
	END_CASE

	//Call to FB Cyclic Logic
	TestFBSimulationSetHMI.CyclicLogic();
END_IF
END_METHOD

METHOD SimulationSetProperty
VAR_INST
	State			: INT;
	ActualResult	: BOOL;
	ActualResultHMI : BOOL;
	ExpectedResult	: BOOL := TRUE;
END_VAR
IF TEST_ORDERED('SimulationSetProperty') THEN
	CASE State OF
		0:
			State := State + 10;

		10:
			IF TestFBSimulationSetProperty.InitComplete AND NOT TestFBSimulationSetProperty.Busy THEN
				State := State + 10;
			END_IF

		20:
			TestFBSimulationSetProperty.InSimulation := TRUE;
			State									 := State + 10;

		30:
			ActualResult	:= TestFBSimulationSetProperty.InSimulation;
			ActualResultHMI := TestFBSimulationSetProperty.ComponentBase_HMI.Status.InSimulation;
			AssertEquals_BOOL(Expected := ExpectedResult, Actual := ActualResult, Message := 'Function Block did not set simulation by property when read by Property');
			AssertEquals_BOOL(Expected := ExpectedResult, Actual := ActualResultHMI, Message := 'Function Block did not set simulation by property when read by HMI');
			TEST_FINISHED();
			State := State + 10;
	END_CASE

	//Call to FB Cyclic Logic
	TestFBSimulationSetProperty.CyclicLogic();
END_IF
END_METHOD

END_FUNCTION_BLOCK

// Testing/Solenoids/FB_DoubleSolenoid_Test
FUNCTION_BLOCK FB_DoubleSolenoid_Test EXTENDS TcUnit.FB_TestSuite
VAR
	TestFBExtend  : FB_DoubleSolenoid;
	TestFBRetract : FB_DoubleSolenoid;
END_VAR

ExtendEqualsExtendOutputOnRetractOff();
RetractEqualsExtendOutputOffRetractOutputOn();

METHOD ExtendEqualsExtendOutputOnRetractOff
VAR_INST
	State						: INT;
	ActualExtendOutputResult	: BOOL;
	ActualRetractOutputResult	: BOOL;
	ExpectedExtendOutputResult	: BOOL := TRUE;
	ExpectedRetractOutputResult : BOOL := FALSE;
END_VAR
IF TEST_ORDERED('ExtendEqualsExtendOutputOnRetractOff') THEN
	CASE State OF
		0:
			State := State + 10;

		10:
			IF TestFBExtend.InitComplete AND NOT TestFBExtend.Busy THEN
				TestFBExtend.Extend();
				State := State + 10;
			END_IF

		20:
			ActualExtendOutputResult := TestFBExtend.ExtendOutput;
			AssertEquals_BOOL(Expected := ExpectedExtendOutputResult, Actual := ActualExtendOutputResult, Message := 'Solenoid did not set extend output on');
			ActualRetractOutputResult := TestFBExtend.RetractOutput;
			AssertEquals_BOOL(Expected := ExpectedRetractOutputResult, Actual := ActualRetractOutputResult, Message := 'Solenoid did not set retract output off');
			TEST_FINISHED();
			State := State + 10;
	END_CASE

	TestFBExtend.CyclicLogic();
END_IF
END_METHOD

METHOD RetractEqualsExtendOutputOffRetractOutputOn
VAR_INST
	State						: INT;
	ActualExtendOutputResult	: BOOL;
	ActualRetractOutputResult	: BOOL;
	ExpectedExtendOutputResult	: BOOL := FALSE;
	ExpectedRetractOutputResult : BOOL := TRUE;
END_VAR
IF TEST_ORDERED('ExtendEqualsExtendOutputOffRetractOn') THEN
	CASE State OF
		0:
			State := State + 10;

		10:
			IF TestFBRetract.InitComplete AND NOT TestFBRetract.Busy THEN
				TestFBRetract.Extend();
				State := State + 10;
			END_IF

		20:
			IF TestFBRetract.Extended THEN
				TestFBRetract.Retract();
				State := State + 10;
			END_IF

		30:
			ActualExtendOutputResult := TestFBRetract.ExtendOutput;
			AssertEquals_BOOL(Expected := ExpectedExtendOutputResult, Actual := ActualExtendOutputResult, Message := 'Solenoid did not set extend output off');
			ActualRetractOutputResult := TestFBRetract.RetractOutput;
			AssertEquals_BOOL(Expected := ExpectedRetractOutputResult, Actual := ActualRetractOutputResult, Message := 'Solenoid did not set retract output on');
			TEST_FINISHED();
			State := State + 10;
	END_CASE

	TestFBRetract.CyclicLogic();
END_IF
END_METHOD

END_FUNCTION_BLOCK

// Testing/Solenoids/FB_SingleSolenoidFeedback_Test
FUNCTION_BLOCK FB_SingleSolenoidFeedback_Test EXTENDS FB_TestSuite
VAR
	// Solenoid FB	
	TestSingleSolenoidFeedbackExtend	   : FB_SingleSolenoidFeedback;
	TestSingleSolenoidFeedbackExtendError  : FB_SingleSolenoidFeedback;
	TestSingleSolenoidFeedbackRetract	   : FB_SingleSolenoidFeedback;
	TestSingleSolenoidFeedbackRetractError : FB_SingleSolenoidFeedback;
END_VAR

Extend();
ExtendError();

METHOD Extend
VAR_INST
	State		   : INT;
	ActualResult   : BOOL;
	ExpectedResult : BOOL := TRUE;
END_VAR
IF TEST_ORDERED('SingleSolenoidFeedbackTestExtend') THEN
	CASE State OF
		0:
			IF TestSingleSolenoidFeedbackExtend.InitComplete AND NOT TestSingleSolenoidFeedbackExtend.Busy THEN
				TestSingleSolenoidFeedbackExtend.Extend();
				TestSingleSolenoidFeedbackExtend.ExtendedInput	:= TRUE;  //Set the feedback
				TestSingleSolenoidFeedbackExtend.RetractedInput := FALSE; //Set the feedback
				State											:= State + 10;
			END_IF

		10:
			ActualResult := TestSingleSolenoidFeedbackExtend.Extended;
			AssertEquals_BOOL(Expected := ExpectedResult, Actual := ActualResult, Message := 'Solenoid feedback did not turn on');
			State := State + 10;
			TEST_FINISHED();
	END_CASE

	TestSingleSolenoidFeedbackExtend.CyclicLogic();
END_IF
END_METHOD

METHOD ExtendError
VAR_INST
	State				: INT;
	ActualResult		: BOOL;
	ExpectedResult		: BOOL := FALSE;
	ActualErrorResult	: BOOL;
	ExpectedErrorResult : BOOL := TRUE;
END_VAR
IF TEST_ORDERED('SingleSolenoidFeedbackTestExtendError') THEN
	CASE State OF
		0:
			IF TestSingleSolenoidFeedbackExtendError.InitComplete AND NOT TestSingleSolenoidFeedbackExtendError.Busy THEN
				TestSingleSolenoidFeedbackExtendError.Extend();
				State := State + 10;
			END_IF

		10:
			IF TestSingleSolenoidFeedbackExtendError.Extended OR TestSingleSolenoidFeedbackExtendError.Error THEN
				ActualResult := TestSingleSolenoidFeedbackExtendError.Extended;
				AssertEquals_BOOL(Expected := ExpectedResult, Actual := ActualResult, Message := 'Solenoid feedback did not turn on');
				ActualErrorResult := TestSingleSolenoidFeedbackExtendError.Error;
				AssertEquals_BOOL(Expected := ExpectedErrorResult, Actual := ActualErrorResult, Message := 'Solenoid Feedback extend no error');
				State := State + 10;
				TEST_FINISHED();
			END_IF
	END_CASE

	TestSingleSolenoidFeedbackExtendError.CyclicLogic();
END_IF
END_METHOD

END_FUNCTION_BLOCK
